# EPICS autosave request: BPMRFFEApp/Db/bpmrffe.req
$(P)$(R)Att-SP
$(P)$(R)PidSpAC-SP
$(P)$(R)PidSpBD-SP
$(P)$(R)TempCtl-SP
$(P)$(R)HeaterAC-SP
$(P)$(R)HeaterBD-SP
$(P)$(R)PidACKp-SP
$(P)$(R)PidACTi-SP
$(P)$(R)PidACTd-SP
$(P)$(R)PidBDKp-SP
$(P)$(R)PidBDTi-SP
$(P)$(R)PidBDTd-SP
